// TIA Portal V18 export
FUNCTION "AIadv" : Void   // FC10013, FBD
{ S7_Optimized_Access := 'TRUE' }
VERSION : 0.1
// stored: AutoNumber false, IsIECCheckEnabled false, SetENOAutomatically false, UDAEnableTagReadback false
   VAR_INPUT
      iInput : Int;
      rFilterValue : Real;
      rMin : Real;
      rMax : Real;
      rCalibration : Real;
   END_VAR
   VAR_OUTPUT
      rOutput : Real;
   END_VAR
   VAR_TEMP
      rNorm : Real;
      rScaled : Real;
      rOut_real : Real;
   END_VAR
   VAR CONSTANT
      iRawMin : Int := 0;
      iRawMax : Int := 27648;
   END_VAR
BEGIN

REGION Network 1 (SCL)
   #rNorm := NORM_X(
                    MIN := #iRawMin,
                    VALUE := #iInput,
                    MAX := #iRawMax);
END_REGION

REGION Network 2 (SCL)
   #rScaled := SCALE_X(
                       MIN := #rMin,
                       VALUE := #rNorm,
                       MAX := #rMax);
END_REGION

REGION Network 3 (SCL): // --- Обмеження межами ---
   IF #rScaled < #rMin THEN
       #rScaled := #rMin;
   ELSIF #rScaled > #rMax THEN
       #rScaled := #rMax;
   END_IF;
END_REGION

REGION Network 4 (SCL): // --- Калібрування (зсув) ---
   #rOutput := #rScaled + #rCalibration;
END_REGION

REGION Network 5 (SCL): // --- Підготовка коеф. фільтра ---
   // rFilterSet = 1.0 → фільтр «прозорий» (швидка реакція, без згладжування).
   // 
   // rFilterSet = 0.1…0.3 → м’яке згладжування.
   // 
   // rFilterSet = 0.0 → вихід «заморожений».
   // --- Підготовка коеф. фільтра ---
   //rAlpha := rFilterSet;/
   //IF rAlpha < 0.0 THEN
   //    rAlpha := 0.0;
   //END_IF;
   //IF rAlpha > 1.0 THEN
   //    rAlpha := 1.0;
   //END_IF;

   // --- Ініціалізація ---
   //IF xInit THEN
   //    rY := rScaledRaw;/
   //    xInit := FALSE;
   //END_IF;

   // --- Фільтр: y = y + α*(x - y) ---
   //rY := rY + rAlpha * (rScaledRaw - rY);

   // --- Вихід ---
   //#rOutput := rY;
END_REGION
END_FUNCTION
